(* PLC project PLC1, Beckhoff Automation GmbH TwinCAT PLC Control 3.5.13.21 *)
(* stored: creationDateTime 2022-08-11T18:58:03.4496374, modificationDateTime 2022-08-11T18:58:03.4496374 *)

FUNCTION_BLOCK FB_Bool_To_Word
VAR_INPUT
	inArrayOfBool : ARRAY [0..15] OF BOOL;
END_VAR
VAR_OUTPUT
	outWord : WORD;
END_VAR
VAR
END_VAR

            outWord.0:=inArrayOfBool[0];
outWord.1:=inArrayOfBool[1];
outWord.2:=inArrayOfBool[2];
outWord.3:=inArrayOfBool[3];
outWord.4:=inArrayOfBool[4];
outWord.5:=inArrayOfBool[5];
outWord.6:=inArrayOfBool[6];
outWord.7:=inArrayOfBool[7];
outWord.8:=inArrayOfBool[8];
outWord.9:=inArrayOfBool[9]; 
outWord.10:=inArrayOfBool[10];
outWord.11:=inArrayOfBool[11];
outWord.12:=inArrayOfBool[12];
outWord.13:=inArrayOfBool[13];
outWord.14:=inArrayOfBool[14];
outWord.15:=inArrayOfBool[15];

          
END_FUNCTION_BLOCK
